PROGRAM MAIN
VAR
END_VAR

END_PROGRAM

(* stored: Version 1.1.0.1
   POU MAIN: Id {25b993f9-81f6-412e-acb0-4d498288e8e2} *)
